ABB RobotStudio station: Montaje_Herramienta.rsstnx

Station Montaje_Herramienta (saved by RobotStudio 23.4.10609.1)
Controller Controlador1
  mechanical unit ROB_1: IRB140_6_81_C_03, 6 joints, base frame (0, 0, 0) mm
Layout (positions relative to the parent item):
  - IRB140_6_81_C_03 [mechanism, from %ABB.RobotStudio.Models.IRB140%\IRB140_6_81_C_G_03.rslib] at (0, 0, 0) mm; joint values [0, 0, 0, 0, 0.5236, 0] (rad or m)
  - Logo_names_45 [part] at (800, 300, 0) mm, rotated rx 0 ry 0 rz 180 deg, size 307.1 x 300 x 219.2 mm
  - MyNewTool [mechanism] at (506.29, 0, 679.5) mm, rotated rx 180 ry 60 rz 180 deg
      TCP MyNewTool at (0, 103.94, 156.44) mm, rotated rx 0 ry 45 rz 90 deg
      links: Support_RS
Attachment: MyNewTool is attached to IRB140_6_81_C_03 / Link6
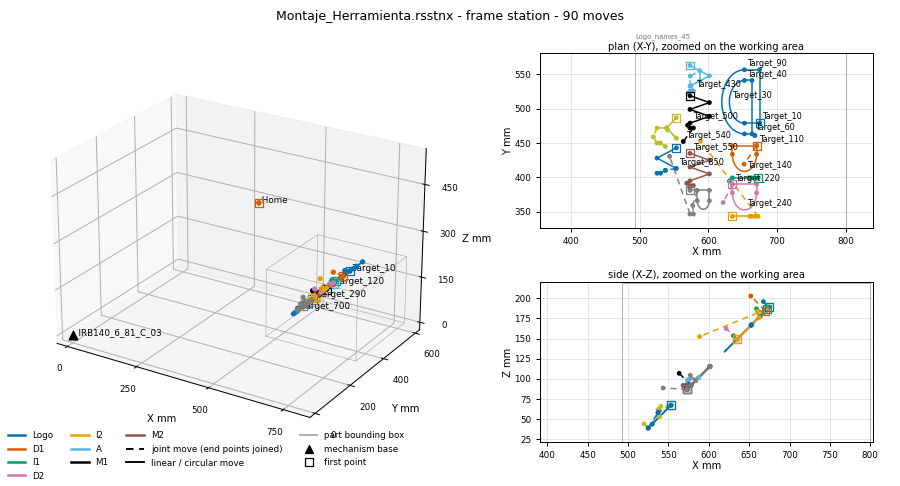
[picture p0: tool path of Montaje_Herramienta.rsstnx in frame station, 90 of 90 moves have a stored position in this frame; points joined in program order, loops and branches not executed]
Targets, tools, work objects and paths stored in the station, written as RAPID:
! task T_ROB1
MODULE CalibData
  TASK PERS wobjdata Workobject_1:=[FALSE,TRUE,"",[[712.132,300,212.132],[0.382683432,0,0.923879533,0]],[[0,0,-10],[1,0,0,0]]];
  PERS tooldata MyNewTool:=[TRUE,[[73.5,73.5,156.444696834],[0.853553391,-0.146446609,0.353553391,0.353553391]],[1,[0,0,1],[1,0,0,0],0,0,0]];
ENDMODULE

! task T_ROB1
MODULE Module1
  CONST robtarget Target_10:=[[43.067,178.883,0],[1,0,0,0],[0,-2,1,0],[9E+09,9E+09,9E+09,9E+09,9E+09,9E+09]];
  CONST robtarget Target_20:=[[74.267,178.883,0],[1,0,0,0],[0,-2,1,0],[9E+09,9E+09,9E+09,9E+09,9E+09,9E+09]];
  CONST robtarget Target_30:=[[105.467,210.083,0],[1,0,0,0],[0,-2,1,0],[9E+09,9E+09,9E+09,9E+09,9E+09,9E+09]];
  CONST robtarget Target_40:=[[74.267,241.283,0],[1,0,0,0],[0,-2,0,0],[9E+09,9E+09,9E+09,9E+09,9E+09,9E+09]];
  CONST robtarget Target_50:=[[58.667,241.283,0],[1,0,0,0],[0,-2,0,0],[9E+09,9E+09,9E+09,9E+09,9E+09,9E+09]];
  CONST robtarget Target_60:=[[58.667,163.283,0],[1,0,0,0],[0,-2,1,0],[9E+09,9E+09,9E+09,9E+09,9E+09,9E+09]];
  CONST robtarget Target_70:=[[74.267,163.283,0],[1,0,0,0],[0,-2,1,0],[9E+09,9E+09,9E+09,9E+09,9E+09,9E+09]];
  CONST robtarget Target_80:=[[121.067,210.083,0],[1,0,0,0],[0,-2,1,0],[9E+09,9E+09,9E+09,9E+09,9E+09,9E+09]];
  CONST robtarget Target_90:=[[74.267,256.883,0],[1,0,0,0],[0,-2,0,0],[9E+09,9E+09,9E+09,9E+09,9E+09,9E+09]];
  CONST robtarget Target_100:=[[43.067,256.883,0],[1,0,0,0],[0,-2,0,0],[9E+09,9E+09,9E+09,9E+09,9E+09,9E+09]];
  CONST robtarget Target_110:=[[49.307,146.077,0],[1,0,0,0],[0,-2,1,0],[9E+09,9E+09,9E+09,9E+09,9E+09,9E+09]];
  CONST robtarget Target_120:=[[99.226985269,146.076975233,0.000011329],[1,0.000000004,0.00000003,-0.000000033],[0,-2,1,0],[9E+09,9E+09,9E+09,9E+09,9E+09,9E+09]];
  CONST robtarget Target_130:=[[99.227,133.597,0],[1,0,0,0],[0,-2,1,0],[9E+09,9E+09,9E+09,9E+09,9E+09,9E+09]];
  CONST robtarget Target_140:=[[74.267,108.637,0],[1,0,0,0],[0,-2,1,0],[9E+09,9E+09,9E+09,9E+09,9E+09,9E+09]];
  CONST robtarget Target_150:=[[49.307,133.597,0],[1,0,0,0],[0,-2,1,0],[9E+09,9E+09,9E+09,9E+09,9E+09,9E+09]];
  CONST robtarget Target_160:=[[46.187,99.277,0],[1,0,0,0],[0,0,0,0],[9E+09,9E+09,9E+09,9E+09,9E+09,9E+09]];
  CONST robtarget Target_170:=[[52.427,99.277,0],[1,0,0,0],[0,-2,1,0],[9E+09,9E+09,9E+09,9E+09,9E+09,9E+09]];
  CONST robtarget Target_180:=[[60.227,99.277,0],[1,0,0,0],[0,-2,1,0],[9E+09,9E+09,9E+09,9E+09,9E+09,9E+09]];
  CONST robtarget Target_190:=[[99.227,99.277,0],[1,0,0,0],[0,-2,1,0],[9E+09,9E+09,9E+09,9E+09,9E+09,9E+09]];
  CONST robtarget Target_200:=[[55.434807347,99.276990865,-9.570120905],[1,-0.000000033,0.000000018,-0.000000049],[0,-2,1,0],[9E+09,9E+09,9E+09,9E+09,9E+09,9E+09]];
  CONST robtarget Target_210:=[[49.307,89.917,0],[1,0,0,0],[0,-2,1,0],[9E+09,9E+09,9E+09,9E+09,9E+09,9E+09]];
  CONST robtarget Target_220:=[[99.227,89.917,0],[1,0,0,0],[0,-2,1,0],[9E+09,9E+09,9E+09,9E+09,9E+09,9E+09]];
  CONST robtarget Target_230:=[[99.227,77.437,0],[1,0,0,0],[0,-2,1,0],[9E+09,9E+09,9E+09,9E+09,9E+09,9E+09]];
  CONST robtarget Target_240:=[[74.267,52.477,0],[1,0,0,0],[0,-2,1,0],[9E+09,9E+09,9E+09,9E+09,9E+09,9E+09]];
  CONST robtarget Target_250:=[[49.307,77.437,0],[1,0,0,0],[0,-2,1,0],[9E+09,9E+09,9E+09,9E+09,9E+09,9E+09]];
  CONST robtarget Target_260:=[[46.187,43.117,0],[1,0,0,0],[0,-2,1,0],[9E+09,9E+09,9E+09,9E+09,9E+09,9E+09]];
  CONST robtarget Target_270:=[[52.427,43.117,0],[1,0,0,0],[0,-2,1,0],[9E+09,9E+09,9E+09,9E+09,9E+09,9E+09]];
  CONST robtarget Target_280:=[[60.227,43.117,0],[1,0,0,0],[0,-2,1,0],[9E+09,9E+09,9E+09,9E+09,9E+09,9E+09]];
  CONST robtarget Target_290:=[[99.227,43.117,0],[1,0,0,0],[0,-2,1,0],[9E+09,9E+09,9E+09,9E+09,9E+09,9E+09]];
  CONST robtarget Target_300:=[[56.841351546,43.117002325,-6.657346861],[1,-0.000000054,0.000000041,0.000000045],[0,-2,1,0],[9E+09,9E+09,9E+09,9E+09,9E+09,9E+09]];
  CONST robtarget Target_310:=[[43.067062574,160.806086079,-9.853973671],[1,-0.00000004,0.000000028,-0.000000016],[0,-2,1,0],[9E+09,9E+09,9E+09,9E+09,9E+09,9E+09]];
  CONST robtarget Target_320:=[[49.307046828,119.23288763,-25.759612298],[1,-0.000000046,0.000000065,-0.00000006],[0,-2,1,0],[9E+09,9E+09,9E+09,9E+09,9E+09,9E+09]];
  CONST robtarget Target_330:=[[99.227222136,94.540167228,-6.232927613],[1,-0.000000004,0.00000006,-0.000000007],[0,-2,1,0],[9E+09,9E+09,9E+09,9E+09,9E+09,9E+09]];
  CONST robtarget Target_340:=[[99.227234739,63.232616482,-18.994122421],[1,-0.000000078,0.000000016,-0.000000084],[0,-2,1,0],[9E+09,9E+09,9E+09,9E+09,9E+09,9E+09]];
  CONST robtarget Target_350:=[[129.667100346,152.744991131,-35.165737418],[1,-0.000000071,0.000000063,0.000000069],[0,-2,1,0],[9E+09,9E+09,9E+09,9E+09,9E+09,9E+09]];
  CONST robtarget Target_360:=[[186.614,263,0],[1,0,0,0],[0,0,0,0],[9E+09,9E+09,9E+09,9E+09,9E+09,9E+09]];
  CONST robtarget Target_370:=[[146.614,248,0],[1,0,0,0],[0,-2,1,0],[9E+09,9E+09,9E+09,9E+09,9E+09,9E+09]];
  CONST robtarget Target_380:=[[186.614,233,0],[1,0,0,0],[0,-2,1,0],[9E+09,9E+09,9E+09,9E+09,9E+09,9E+09]];
  CONST robtarget Target_390:=[[166.614,255.5,0],[1,0,0,0],[0,-2,1,0],[9E+09,9E+09,9E+09,9E+09,9E+09,9E+09]];
  CONST robtarget Target_400:=[[166.614,240.5,0],[1,0,0,0],[0,-2,1,0],[9E+09,9E+09,9E+09,9E+09,9E+09,9E+09]];
  CONST robtarget Target_410:=[[178.412389788,247.495688741,-7.683915859],[1,0.000000028,0.000000061,-0.000000021],[0,-2,1,0],[9E+09,9E+09,9E+09,9E+09,9E+09,9E+09]];
  CONST robtarget Target_420:=[[177.268953329,233.762683131,-7.389857689],[1,-0.000000071,0.000000053,-0.000000025],[0,-2,1,0],[9E+09,9E+09,9E+09,9E+09,9E+09,9E+09]];
  CONST robtarget Target_430:=[[179.614,226,0],[1,0,0,0],[0,-2,1,0],[9E+09,9E+09,9E+09,9E+09,9E+09,9E+09]];
  CONST robtarget Target_440:=[[186.614,226,0],[1,0,0,0],[0,-2,1,0],[9E+09,9E+09,9E+09,9E+09,9E+09,9E+09]];
  CONST robtarget Target_450:=[[186.614060293,222.892156445,-2.542651344],[1,-0.000000085,0.00000005,-0.000000036],[0,-2,1,0],[9E+09,9E+09,9E+09,9E+09,9E+09,9E+09]];
  CONST robtarget Target_460:=[[186.614,219,0],[1,0,0,0],[0,0,0,0],[9E+09,9E+09,9E+09,9E+09,9E+09,9E+09]];
  CONST robtarget Target_470:=[[146.614,209,0],[1,0,0,0],[0,-2,1,0],[9E+09,9E+09,9E+09,9E+09,9E+09,9E+09]];
  CONST robtarget Target_480:=[[186.614,199,0],[1,0,0,0],[0,-2,1,0],[9E+09,9E+09,9E+09,9E+09,9E+09,9E+09]];
  CONST robtarget Target_490:=[[146.614,189,0],[1,0,0,0],[0,-2,1,0],[9E+09,9E+09,9E+09,9E+09,9E+09,9E+09]];
  CONST robtarget Target_500:=[[186.614,179,0],[1,0,0,0],[0,-2,1,0],[9E+09,9E+09,9E+09,9E+09,9E+09,9E+09]];
  CONST robtarget Target_510:=[[186.614,172,0],[1,0,0,0],[0,-2,1,0],[9E+09,9E+09,9E+09,9E+09,9E+09,9E+09]];
  CONST robtarget Target_520:=[[179.614,172,0],[1,0,0,0],[0,-2,1,0],[9E+09,9E+09,9E+09,9E+09,9E+09,9E+09]];
  CONST robtarget Target_530:=[[186.614131871,175.925884496,-4.92195742],[1,-0.000000022,0.000000055,-0.000000082],[0,-2,1,0],[9E+09,9E+09,9E+09,9E+09,9E+09,9E+09]];
  CONST robtarget Target_540:=[[179.614119452,152.268392323,-20.819936774],[1,-0.000000012,0.000000036,0.000000018],[0,-2,1,0],[9E+09,9E+09,9E+09,9E+09,9E+09,9E+09]];
  CONST robtarget Target_550:=[[186.614,135,0],[1,0,0,0],[0,0,0,0],[9E+09,9E+09,9E+09,9E+09,9E+09,9E+09]];
  CONST robtarget Target_560:=[[146.614,125,0],[1,0,0,0],[0,-2,1,0],[9E+09,9E+09,9E+09,9E+09,9E+09,9E+09]];
  CONST robtarget Target_570:=[[186.614,115,0],[1,0,0,0],[0,-2,1,0],[9E+09,9E+09,9E+09,9E+09,9E+09,9E+09]];
  CONST robtarget Target_580:=[[146.614,105,0],[1,0,0,0],[0,-2,1,0],[9E+09,9E+09,9E+09,9E+09,9E+09,9E+09]];
  CONST robtarget Target_590:=[[186.614,95,0],[1,0,0,0],[0,-2,1,0],[9E+09,9E+09,9E+09,9E+09,9E+09,9E+09]];
  CONST robtarget Target_600:=[[186.614,88,0],[1,0,0,0],[0,-2,1,0],[9E+09,9E+09,9E+09,9E+09,9E+09,9E+09]];
  CONST robtarget Target_610:=[[179.614,88,0],[1,0,0,0],[0,-2,1,0],[9E+09,9E+09,9E+09,9E+09,9E+09,9E+09]];
  CONST robtarget Target_620:=[[186.614151743,91.364782311,-6.75911763],[1,-0.00000011,0.000000243,0.000000801],[0,-2,1,0],[9E+09,9E+09,9E+09,9E+09,9E+09,9E+09]];
  CONST robtarget Target_630:=[[182.85629019,84.770816683,-4.125906462],[1,0.000000024,0.000000045,0.000000006],[0,-2,1,0],[9E+09,9E+09,9E+09,9E+09,9E+09,9E+09]];
  CONST robtarget Target_640:=[[186.614,81,0],[1,0,0,0],[0,0,0,0],[9E+09,9E+09,9E+09,9E+09,9E+09,9E+09]];
  CONST robtarget Target_650:=[[146.614,81,0],[1,0,0,0],[0,-2,1,0],[9E+09,9E+09,9E+09,9E+09,9E+09,9E+09]];
  CONST robtarget Target_660:=[[146.614,66,0],[1,0,0,0],[0,-2,1,0],[9E+09,9E+09,9E+09,9E+09,9E+09,9E+09]];
  CONST robtarget Target_670:=[[159.114,53.5,0],[1,0,0,0],[0,-2,1,0],[9E+09,9E+09,9E+09,9E+09,9E+09,9E+09]];
  CONST robtarget Target_680:=[[171.614,66,0],[1,0,0,0],[0,-2,1,0],[9E+09,9E+09,9E+09,9E+09,9E+09,9E+09]];
  CONST robtarget Target_690:=[[171.614,81,0],[1,0,0,0],[0,-2,1,0],[9E+09,9E+09,9E+09,9E+09,9E+09,9E+09]];
  CONST robtarget Target_700:=[[179.614,46.5,0],[1,0,0,0],[0,-2,1,0],[9E+09,9E+09,9E+09,9E+09,9E+09,9E+09]];
  CONST robtarget Target_710:=[[186.614,46.5,0],[1,0,0,0],[0,-2,1,0],[9E+09,9E+09,9E+09,9E+09,9E+09,9E+09]];
  CONST robtarget Target_720:=[[171.614157585,58.991205559,-9.389654006],[1,-0.000000034,0.000000051,-0.000000007],[0,-2,1,0],[9E+09,9E+09,9E+09,9E+09,9E+09,9E+09]];
  CONST robtarget Target_730:=[[206.575840133,130.575387227,-22.08903626],[1,-0.000000061,0.000000016,-0.000000213],[0,-2,1,0],[9E+09,9E+09,9E+09,9E+09,9E+09,9E+09]];
  CONST robtarget Target_740:=[[214.649,187,0],[1,0,0,0],[0,0,0,0],[9E+09,9E+09,9E+09,9E+09,9E+09,9E+09]];
  CONST robtarget Target_750:=[[234.649,172,0],[1,0,0,0],[0,-2,1,0],[9E+09,9E+09,9E+09,9E+09,9E+09,9E+09]];
  CONST robtarget Target_760:=[[214.649,157,0],[1,0,0,0],[0,-2,1,0],[9E+09,9E+09,9E+09,9E+09,9E+09,9E+09]];
  CONST robtarget Target_770:=[[254.649,172,0],[1,0,0,0],[0,-2,1,0],[9E+09,9E+09,9E+09,9E+09,9E+09,9E+09]];
  CONST robtarget Target_780:=[[247.649,150,0],[1,0,0,0],[0,-2,1,0],[9E+09,9E+09,9E+09,9E+09,9E+09,9E+09]];
  CONST robtarget Target_790:=[[254.649,150,0],[1,0,0,0],[0,-2,1,0],[9E+09,9E+09,9E+09,9E+09,9E+09,9E+09]];
  CONST robtarget Target_800:=[[224.45405819,169.052593882,-7.938534661],[1,-0.000000024,0.000000053,-0.000000097],[0,-2,1,0],[9E+09,9E+09,9E+09,9E+09,9E+09,9E+09]];
  CONST robtarget Target_810:=[[254.649339406,159.007770374,-7.41636934],[1,-0.000000027,0.000000051,-0.000000098],[0,-2,1,0],[9E+09,9E+09,9E+09,9E+09,9E+09,9E+09]];
  CONST robtarget Target_820:=[[229.743212618,145.004792826,-7.759407548],[1,-0.000000014,0.000000023,0.000000082],[0,-2,1,0],[9E+09,9E+09,9E+09,9E+09,9E+09,9E+09]];
  CONST robtarget Target_830:=[[214.649,143,0],[1,0,0,0],[0,0,0,0],[9E+09,9E+09,9E+09,9E+09,9E+09,9E+09]];
  CONST robtarget Target_840:=[[254.649,128,0],[1,0,0,0],[0,-2,1,0],[9E+09,9E+09,9E+09,9E+09,9E+09,9E+09]];
  CONST robtarget Target_850:=[[214.649,113,0],[1,0,0,0],[0,-2,1,0],[9E+09,9E+09,9E+09,9E+09,9E+09,9E+09]];
  CONST robtarget Target_860:=[[247.649,106,0],[1,0,0,0],[0,-2,1,0],[9E+09,9E+09,9E+09,9E+09,9E+09,9E+09]];
  CONST robtarget Target_870:=[[254.649,106,0],[1,0,0,0],[0,-2,1,0],[9E+09,9E+09,9E+09,9E+09,9E+09,9E+09]];
  CONST robtarget Target_880:=[[232.237810088,110.203687427,-5.065784914],[1,-0.000000178,0.000000032,0.000000095],[0,-2,1,0],[9E+09,9E+09,9E+09,9E+09,9E+09,9E+09]];
  CONST robtarget Home:=[[605.026732992,73.5,537.624784405],[0.120590477,0.232962914,0.915975615,0.303603179],[-1,0,-1,0],[9E+09,9E+09,9E+09,9E+09,9E+09,9E+09]];
  PROC Logo()
    MoveJ Target_10,v400,z10,MyNewTool\WObj:=Workobject_1;
    MoveL Target_20,v200,z5,MyNewTool\WObj:=Workobject_1;
    MoveC Target_30,Target_40,v200,z5,MyNewTool\WObj:=Workobject_1;
    MoveL Target_50,v200,z5,MyNewTool\WObj:=Workobject_1;
    MoveL Target_60,v200,z5,MyNewTool\WObj:=Workobject_1;
    MoveL Target_70,v200,z5,MyNewTool\WObj:=Workobject_1;
    MoveC Target_80,Target_90,v200,z5,MyNewTool\WObj:=Workobject_1;
    MoveL Target_100,v200,z5,MyNewTool\WObj:=Workobject_1;
    MoveL Target_10,v200,z5,MyNewTool\WObj:=Workobject_1;
    MoveJ Target_310,v400,z10,MyNewTool\WObj:=Workobject_1;
  ENDPROC
  PROC D1()
    MoveJ Target_110,v400,z10,MyNewTool\WObj:=Workobject_1;
    MoveL Target_120,v400,z10,MyNewTool\WObj:=Workobject_1;
    MoveL Target_130,v200,z5,MyNewTool\WObj:=Workobject_1;
    MoveC Target_140,Target_150,v200,z5,MyNewTool\WObj:=Workobject_1;
    MoveL Target_110,v200,z5,MyNewTool\WObj:=Workobject_1;
    MoveJ Target_320,v400,z10,MyNewTool\WObj:=Workobject_1;
  ENDPROC
  PROC I1()
    MoveJ Target_160,v400,z10,MyNewTool\WObj:=Workobject_1;
    MoveL Target_170,v200,z5,MyNewTool\WObj:=Workobject_1;
    MoveJ Target_200,v400,z10,MyNewTool\WObj:=Workobject_1;
    MoveJ Target_180,v400,z10,MyNewTool\WObj:=Workobject_1;
    MoveL Target_190,v200,z5,MyNewTool\WObj:=Workobject_1;
    MoveJ Target_330,v400,z10,MyNewTool\WObj:=Workobject_1;
  ENDPROC
  PROC D2()
    MoveJ Target_220,v400,z10,MyNewTool\WObj:=Workobject_1;
    MoveL Target_230,v200,z5,MyNewTool\WObj:=Workobject_1;
    MoveC Target_240,Target_250,v200,z5,MyNewTool\WObj:=Workobject_1;
    MoveL Target_210,v200,z5,MyNewTool\WObj:=Workobject_1;
    MoveL Target_220,v200,z5,MyNewTool\WObj:=Workobject_1;
    MoveJ Target_340,v400,z10,MyNewTool\WObj:=Workobject_1;
  ENDPROC
  PROC I2()
    MoveJ Target_290,v400,z10,MyNewTool\WObj:=Workobject_1;
    MoveL Target_280,v200,z5,MyNewTool\WObj:=Workobject_1;
    MoveJ Target_300,v400,z10,MyNewTool\WObj:=Workobject_1;
    MoveJ Target_270,v400,z10,MyNewTool\WObj:=Workobject_1;
    MoveL Target_260,v200,z5,MyNewTool\WObj:=Workobject_1;
    MoveJ Target_350,v400,z10,MyNewTool\WObj:=Workobject_1;
  ENDPROC
  PROC A()
    MoveJ Target_360,v400,z10,MyNewTool\WObj:=Workobject_1;
    MoveL Target_370,v200,z5,MyNewTool\WObj:=Workobject_1;
    MoveL Target_380,v200,z5,MyNewTool\WObj:=Workobject_1;
    MoveJ Target_410,v400,z10,MyNewTool\WObj:=Workobject_1;
    MoveJ Target_390,v400,z10,MyNewTool\WObj:=Workobject_1;
    MoveL Target_400,v200,z5,MyNewTool\WObj:=Workobject_1;
    MoveJ Target_420,v400,z10,MyNewTool\WObj:=Workobject_1;
    MoveJ Target_430,v400,z10,MyNewTool\WObj:=Workobject_1;
    MoveL Target_440,v200,z5,MyNewTool\WObj:=Workobject_1;
    MoveJ Target_450,v400,z10,MyNewTool\WObj:=Workobject_1;
  ENDPROC
  PROC M1()
    MoveJ Target_460,v400,z10,MyNewTool\WObj:=Workobject_1;
    MoveL Target_470,v200,z5,MyNewTool\WObj:=Workobject_1;
    MoveL Target_480,v200,z5,MyNewTool\WObj:=Workobject_1;
    MoveL Target_490,v200,z5,MyNewTool\WObj:=Workobject_1;
    MoveL Target_500,v200,z5,MyNewTool\WObj:=Workobject_1;
    MoveJ Target_530,v400,z10,MyNewTool\WObj:=Workobject_1;
    MoveJ Target_510,v400,z10,MyNewTool\WObj:=Workobject_1;
    MoveL Target_520,v200,z5,MyNewTool\WObj:=Workobject_1;
    MoveJ Target_540,v400,z10,MyNewTool\WObj:=Workobject_1;
  ENDPROC
  PROC M2()
    MoveJ Target_550,v400,z10,MyNewTool\WObj:=Workobject_1;
    MoveL Target_560,v200,z5,MyNewTool\WObj:=Workobject_1;
    MoveL Target_570,v200,z5,MyNewTool\WObj:=Workobject_1;
    MoveL Target_580,v200,z5,MyNewTool\WObj:=Workobject_1;
    MoveL Target_590,v200,z5,MyNewTool\WObj:=Workobject_1;
    MoveJ Target_620,v400,z10,MyNewTool\WObj:=Workobject_1;
    MoveJ Target_600,v400,z10,MyNewTool\WObj:=Workobject_1;
    MoveL Target_610,v200,z5,MyNewTool\WObj:=Workobject_1;
    MoveJ Target_630,v400,z10,MyNewTool\WObj:=Workobject_1;
  ENDPROC
  PROC P()
    MoveJ Target_640,v400,z10,MyNewTool\WObj:=Workobject_1;
    MoveL Target_650,v200,z5,MyNewTool\WObj:=Workobject_1;
    MoveL Target_660,v200,z5,MyNewTool\WObj:=Workobject_1;
    MoveC Target_670,Target_680,v200,z5,MyNewTool\WObj:=Workobject_1;
    MoveL Target_690,v200,z5,MyNewTool\WObj:=Workobject_1;
    MoveJ Target_720,v400,z10,MyNewTool\WObj:=Workobject_1;
    MoveJ Target_700,v400,z10,MyNewTool\WObj:=Workobject_1;
    MoveL Target_710,v200,z5,MyNewTool\WObj:=Workobject_1;
    MoveJ Target_730,v400,z10,MyNewTool\WObj:=Workobject_1;
  ENDPROC
  PROC Y()
    MoveJ Target_740,v400,z10,MyNewTool\WObj:=Workobject_1;
    MoveL Target_750,v200,z5,MyNewTool\WObj:=Workobject_1;
    MoveL Target_760,v200,z5,MyNewTool\WObj:=Workobject_1;
    MoveJ Target_800,v400,z10,MyNewTool\WObj:=Workobject_1;
    MoveJ Target_750,v400,z10,MyNewTool\WObj:=Workobject_1;
    MoveL Target_770,v200,z5,MyNewTool\WObj:=Workobject_1;
    MoveJ Target_810,v400,z10,MyNewTool\WObj:=Workobject_1;
    MoveJ Target_790,v400,z10,MyNewTool\WObj:=Workobject_1;
    MoveL Target_780,v200,z5,MyNewTool\WObj:=Workobject_1;
    MoveJ Target_820,v400,z10,MyNewTool\WObj:=Workobject_1;
  ENDPROC
  PROC V()
    MoveJ Target_830,v400,z10,MyNewTool\WObj:=Workobject_1;
    MoveL Target_840,v200,z5,MyNewTool\WObj:=Workobject_1;
    MoveL Target_850,v200,z5,MyNewTool\WObj:=Workobject_1;
    MoveJ Target_880,v400,z10,MyNewTool\WObj:=Workobject_1;
    MoveJ Target_860,v400,z10,MyNewTool\WObj:=Workobject_1;
    MoveL Target_870,v200,z5,MyNewTool\WObj:=Workobject_1;
    MoveJ Target_880,v400,z10,MyNewTool\WObj:=Workobject_1;
  ENDPROC
  PROC Main()
    MoveJ Home,v400,z10,MyNewTool\WObj:=wobj0;
    Logo;
    D1;
    I1;
    D2;
    I2;
    A;
    M1;
    M2;
    P;
    Y;
    V;
    MoveJ Home,v400,z10,MyNewTool\WObj:=wobj0;
  ENDPROC
ENDMODULE

